{attribute 'qualified_only'}
{attribute 'strict'}
TYPE E_DataSequence :
(	
	//E_Send,
	//E_SendWait,
	//E_Recieve,
	//E_RecieveWait
	DUMMY
);
END_TYPE

(* stored: Version 1.1.0.1
   DUT E_DataSequence: Id {78c9dff4-e8e0-4e89-97f2-63c140b1ff91} *)
